// TwinCAT 3 PLC project OPC
// ProgramVersion: 3.1.4023.0
// libraries:
//   Tc2_Standard, * (Beckhoff Automation GmbH)
//   Tc2_System, * (Beckhoff Automation GmbH)
//   Tc3_Module, * (Beckhoff Automation GmbH)
// project tree:
//   GVLs/ dbIO.TcGVL
//   / PlcTask.TcTTO
//   POUs/ fbRaiseTemperature.TcPOU, MAIN.TcPOU
// real-time tasks:
//   TASK PlcTask: cycle T#10ms, priority 20, ADS port 350
//   TASK Device 1 (OPC UA Virtual)_Task_58: cycle T#40ms, priority 58, ADS port 351
// I/O:
//   DEVICE Device 1 (OPC UA Virtual), AmsNetId 192.168.1.207.2.1
// variable links:
//   OPC/OPC Instance <-> Device 1 (OPC UA Virtual)/Client #1
//     PlcTask Outputs/dbIO.bWriteEnable <-> Outputs/Control/Write Enable
//   OPC/OPC Instance <-> Device 1 (OPC UA Virtual)/Client #1/Machine.Alarm
//     PlcTask Outputs/dbIO.bAlarm <-> Outputs/Value
//   OPC/OPC Instance <-> Device 1 (OPC UA Virtual)/Client #1/Machine.Reset
//     PlcTask Inputs/dbIO.bReset <-> Inputs/Value
//   OPC/OPC Instance <-> Device 1 (OPC UA Virtual)/Client #1/Machine.Temperature
//     PlcTask Outputs/dbIO.rTemperature <-> Outputs/Value

CONFIGURATION OPC
    RESOURCE PLC ON TwinCAT3
        TASK PlcTask(INTERVAL := T#10ms, PRIORITY := 20);
        PROGRAM MAIN WITH PlcTask : MAIN;
    END_RESOURCE
END_CONFIGURATION

// ---- GVLs/dbIO.TcGVL
{attribute 'qualified_only'}
VAR_GLOBAL
	bReset  	 AT %I* : BOOL;
	bAlarm  	 AT %Q* : BOOL;
	bWriteEnable AT %Q* : BOOL;
	rTemperature AT %Q* : LREAL;
END_VAR

// ---- POUs/MAIN.TcPOU
PROGRAM MAIN
VAR
	pTemperature : fbRaiseTemperature;
END_VAR


dbIO.bWriteEnable:=TRUE;

pTemperature(bReset := dbIO.bReset,
			bAlarm => dbIO.bAlarm,
			rTemperature => dbIO.rTemperature);

END_PROGRAM

// ---- POUs/fbRaiseTemperature.TcPOU
FUNCTION_BLOCK fbRaiseTemperature
VAR_INPUT
	bReset: BOOL;
END_VAR
VAR_OUTPUT
	bAlarm: BOOL;
	rTemperature: REAL;
END_VAR
VAR
	timer: ton;
END_VAR


timer(PT:=T#1S);

IF NOT Timer.Q AND NOT timer.IN THEN
	timer.IN:=TRUE;
END_IF
 

IF bReset THEN
	timer.IN:=FALSE;
	rTemperature:=0;
	bAlarm:=FALSE;
	timer.IN :=TRUE;
END_IF

IF timer.Q THEN
	timer.IN:=FALSE;
	rTemperature:= rTemperature +1;
END_IF

IF rTemperature >19 THEN
	bAlarm :=TRUE;
END_IF

END_FUNCTION_BLOCK
